SYSTEM DASDA1_27 (* System Configuration *)
  (* Standard: 61499-1 *)
  (* Version 0.4, 2009-03-05, JHC, Holobloc Inc., Deleted Application. *)
  (* Version 0.3, 2003-12-05, JHC, Rockwell Automation, Renamed from NEWSYSTEM. *)
  (* Version 0.2, 2002-11-05, JHC, Rockwell Automation, Fixed missing (empty) FBD in Application. *)
  (* Version 0.1, 2002-01-17, JHC, Rockwell Automation, Minor cleanup *)
  (* Version 0.0, 2000-05-27, JHC, Rockwell Automation *)
  DEVICE HMI_LAYER : FRAME_DEVICE(BOUNDS := [0,0,200,600])
    RESOURCE HMI_left : PANEL_RESOURCE(COLS := 1, ROWS := 10)
      FBS
        start2 : PUBL_0;
        greenTime2 : IN_ANY(TYPE := "UINT", QI := 1, IVAL := "5");
        yellowTime2 : IN_ANY(QI := 1, TYPE := "UINT", IVAL := "1");
        times2 : PUBL_2;
        LABEL1 : FB_LABEL(LABEL := "Western lights control", QI := 1);
        LABEL2 : FB_LABEL(LABEL := "Green time", QI := 1);
        LABEL3 : FB_LABEL(LABEL := "Yellow time", QI := 1);
        minGreenTime2 : IN_ANY(TYPE := "UINT", QI := 1, IVAL := "3");
        LABEL4 : FB_LABEL(LABEL := "Minimum green time", QI := 1);
        Walker1 : IN_EVENT(LABEL := "Walker", QI := 1);
        WalkerTimes2 : PUBL_1;
        RoadControl1 : SUBL_0;
        permit2 : E_PERMIT;
        setreset2 : E_SR;
        split1 : E_SPLIT;
        RoadControl2 : SUBL_0;
        pressCounter : E_CTD(PV := 4);
        split3 : E_SPLIT;
        split4 : E_SPLIT;
        select1 : E_SEL_UINT;
        PedestrianControl2 : SUBL_0;
        gdelay : E_DELAY(DT := t#4000ms);
        setreset3 : E_SR;
        and : FB_AND;
        merge3 : E_MERGE;
        gtrig : E_TRIG;
      END_FBS
      EVENT_CONNECTIONS
        yellowTime2.IND TO times2.REQ;
        LABEL1.INITO TO LABEL2.INIT;
        LABEL2.INITO TO greenTime2.INIT;
        greenTime2.INITO TO LABEL4.INIT;
        LABEL4.INITO TO minGreenTime2.INIT;
        greenTime2.IND TO yellowTime2.REQ;
        yellowTime2.INITO TO times2.INIT;
        times2.INITO TO start2.INIT;
        times2.CNF TO start2.REQ;
        minGreenTime2.INITO TO Walker1.INIT;
        Walker1.INITO TO LABEL3.INIT;
        LABEL3.INITO TO yellowTime2.INIT;
        start2.INITO TO WalkerTimes2.INIT;
        START.COLD TO RoadControl1.INIT;
        RoadControl1.IND TO split1.EI;
        RoadControl2.IND TO setreset2.R;
        RoadControl1.INITO TO RoadControl2.INIT;
        RoadControl2.INITO TO LABEL1.INIT;
        split4.EO1 TO setreset2.S;
        Walker1.IND TO permit2.EI;
        permit2.EO TO split3.EI;
        split3.EO1 TO minGreenTime2.REQ;
        minGreenTime2.IND TO select1.EI0;
        select1.EO TO WalkerTimes2.REQ;
        split4.EO2 TO pressCounter.LD;
        split3.EO2 TO pressCounter.CD;
        PedestrianControl2.IND TO gdelay.START;
        gdelay.EO TO setreset3.S;
        setreset3.EO TO merge3.EI1;
        pressCounter.CDO TO merge3.EI2;
        merge3.EO TO and.REQ;
        and.CNF TO gtrig.EI;
        gtrig.ER TO select1.EI1;
        gtrig.EF TO setreset3.R;
        split1.EO1 TO greenTime2.REQ;
        split1.EO2 TO split4.EI;
        WalkerTimes2.INITO TO PedestrianControl2.INIT;
      END_CONNECTIONS
      DATA_CONNECTIONS
        yellowTime2.OUT TO times2.SD_2;
        greenTime2.OUT TO times2.SD_1;
        setreset2.Q TO permit2.PERMIT;
        minGreenTime2.OUT TO select1.IN0;
        select1.OUT TO WalkerTimes2.SD_1;
        pressCounter.CV TO select1.IN1;
        setreset3.Q TO and.IN1;
        pressCounter.Q TO and.IN2;
        and.OUT TO gtrig.QI;
      END_CONNECTIONS
    END_RESOURCE
    RESOURCE HMI_up : PANEL_RESOURCE(COLS := 1, ROWS := 10)
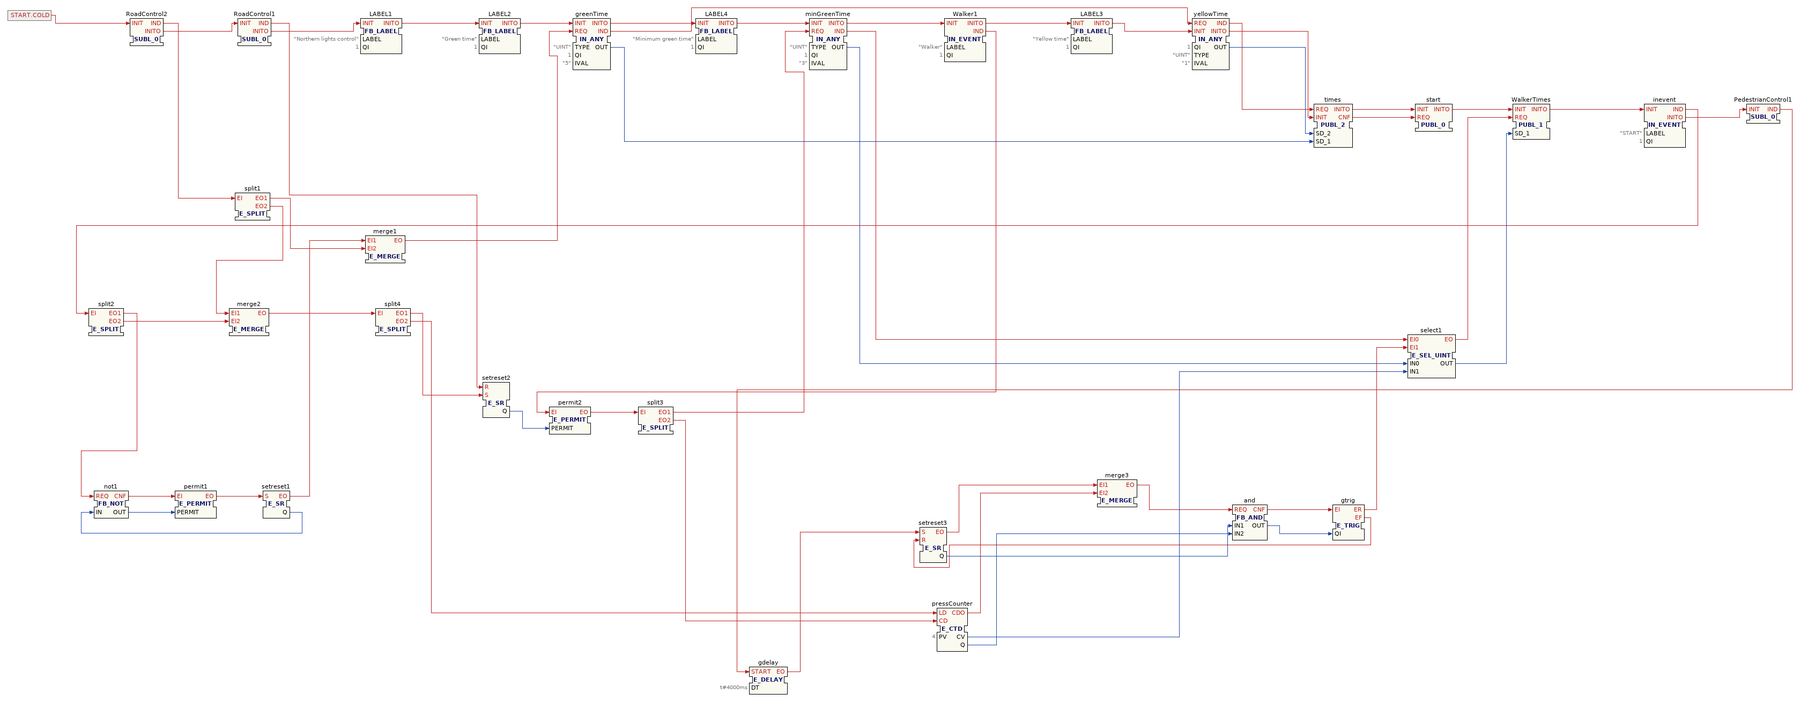
      FBS
        start : PUBL_0;
        greenTime : IN_ANY(TYPE := "UINT", QI := 1, IVAL := "5");
        yellowTime : IN_ANY(QI := 1, TYPE := "UINT", IVAL := "1");
        times : PUBL_2;
        LABEL1 : FB_LABEL(LABEL := "Northern lights control", QI := 1);
        LABEL2 : FB_LABEL(LABEL := "Green time", QI := 1);
        LABEL3 : FB_LABEL(LABEL := "Yellow time", QI := 1);
        minGreenTime : IN_ANY(TYPE := "UINT", QI := 1, IVAL := "3");
        LABEL4 : FB_LABEL(LABEL := "Minimum green time", QI := 1);
        Walker1 : IN_EVENT(LABEL := "Walker", QI := 1);
        WalkerTimes : PUBL_1;
        inevent : IN_EVENT(LABEL := "START", QI := 1);
        RoadControl2 : SUBL_0;
        merge1 : E_MERGE;
        permit1 : E_PERMIT;
        setreset1 : E_SR;
        not1 : FB_NOT;
        permit2 : E_PERMIT;
        setreset2 : E_SR;
        split1 : E_SPLIT;
        RoadControl1 : SUBL_0;
        merge2 : E_MERGE;
        split2 : E_SPLIT;
        pressCounter : E_CTD(PV := 4);
        split3 : E_SPLIT;
        split4 : E_SPLIT;
        select1 : E_SEL_UINT;
        PedestrianControl1 : SUBL_0;
        gdelay : E_DELAY(DT := t#4000ms);
        setreset3 : E_SR;
        and : FB_AND;
        merge3 : E_MERGE;
        gtrig : E_TRIG;
      END_FBS
      EVENT_CONNECTIONS
        yellowTime.IND TO times.REQ;
        LABEL1.INITO TO LABEL2.INIT;
        LABEL2.INITO TO greenTime.INIT;
        greenTime.INITO TO LABEL4.INIT;
        LABEL4.INITO TO minGreenTime.INIT;
        greenTime.IND TO yellowTime.REQ;
        yellowTime.INITO TO times.INIT;
        times.INITO TO start.INIT;
        times.CNF TO start.REQ;
        minGreenTime.INITO TO Walker1.INIT;
        Walker1.INITO TO LABEL3.INIT;
        LABEL3.INITO TO yellowTime.INIT;
        start.INITO TO WalkerTimes.INIT;
        merge1.EO TO greenTime.REQ;
        not1.CNF TO permit1.EI;
        permit1.EO TO setreset1.S;
        setreset1.EO TO merge1.EI1;
        START.COLD TO RoadControl2.INIT;
        WalkerTimes.INITO TO inevent.INIT;
        RoadControl2.IND TO split1.EI;
        split1.EO1 TO merge1.EI2;
        RoadControl1.IND TO setreset2.R;
        RoadControl2.INITO TO RoadControl1.INIT;
        RoadControl1.INITO TO LABEL1.INIT;
        split1.EO2 TO merge2.EI1;
        inevent.IND TO split2.EI;
        split2.EO1 TO not1.REQ;
        split2.EO2 TO merge2.EI2;
        merge2.EO TO split4.EI;
        split4.EO1 TO setreset2.S;
        Walker1.IND TO permit2.EI;
        permit2.EO TO split3.EI;
        split3.EO1 TO minGreenTime.REQ;
        minGreenTime.IND TO select1.EI0;
        select1.EO TO WalkerTimes.REQ;
        split4.EO2 TO pressCounter.LD;
        split3.EO2 TO pressCounter.CD;
        inevent.INITO TO PedestrianControl1.INIT;
        PedestrianControl1.IND TO gdelay.START;
        gdelay.EO TO setreset3.S;
        setreset3.EO TO merge3.EI1;
        pressCounter.CDO TO merge3.EI2;
        merge3.EO TO and.REQ;
        and.CNF TO gtrig.EI;
        gtrig.ER TO select1.EI1;
        gtrig.EF TO setreset3.R;
      END_CONNECTIONS
      DATA_CONNECTIONS
        yellowTime.OUT TO times.SD_2;
        greenTime.OUT TO times.SD_1;
        not1.OUT TO permit1.PERMIT;
        setreset1.Q TO not1.IN;
        setreset2.Q TO permit2.PERMIT;
        minGreenTime.OUT TO select1.IN0;
        select1.OUT TO WalkerTimes.SD_1;
        pressCounter.CV TO select1.IN1;
        setreset3.Q TO and.IN1;
        pressCounter.Q TO and.IN2;
        and.OUT TO gtrig.QI;
      END_CONNECTIONS
    END_RESOURCE
  END_DEVICE
  DEVICE MODEL_LAYER : FRAME_DEVICE
    RESOURCE LIGHTS_U : PANEL_RESOURCE
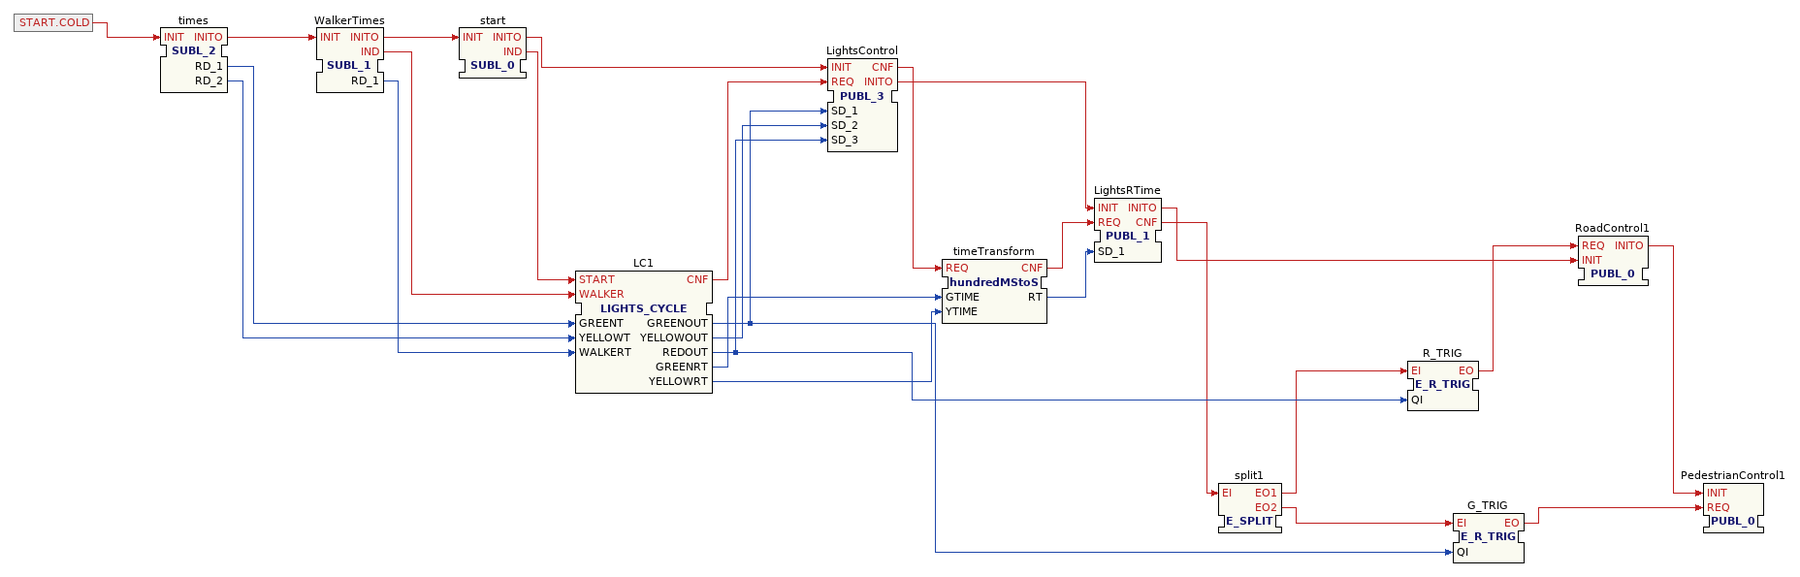
      FBS
        LightsControl : PUBL_3;
        start : SUBL_0;
        times : SUBL_2;
        WalkerTimes : SUBL_1;
        LC1 : LIGHTS_CYCLE;
        R_TRIG : E_R_TRIG;
        RoadControl1 : PUBL_0;
        timeTransform : hundredMStoS;
        LightsRTime : PUBL_1;
        G_TRIG : E_R_TRIG;
        PedestrianControl1 : PUBL_0;
        split1 : E_SPLIT;
      END_FBS
      EVENT_CONNECTIONS
        START.COLD TO times.INIT;
        start.INITO TO LightsControl.INIT;
        times.INITO TO WalkerTimes.INIT;
        WalkerTimes.INITO TO start.INIT;
        start.IND TO LC1.START;
        WalkerTimes.IND TO LC1.WALKER;
        LC1.CNF TO LightsControl.REQ;
        R_TRIG.EO TO RoadControl1.REQ;
        LightsControl.CNF TO timeTransform.REQ;
        LightsControl.INITO TO LightsRTime.INIT;
        LightsRTime.INITO TO RoadControl1.INIT;
        timeTransform.CNF TO LightsRTime.REQ;
        RoadControl1.INITO TO PedestrianControl1.INIT;
        G_TRIG.EO TO PedestrianControl1.REQ;
        LightsRTime.CNF TO split1.EI;
        split1.EO1 TO R_TRIG.EI;
        split1.EO2 TO G_TRIG.EI;
      END_CONNECTIONS
      DATA_CONNECTIONS
        WalkerTimes.RD_1 TO LC1.WALKERT;
        times.RD_1 TO LC1.GREENT;
        times.RD_2 TO LC1.YELLOWT;
        LC1.GREENOUT TO LightsControl.SD_1;
        LC1.YELLOWOUT TO LightsControl.SD_2;
        LC1.REDOUT TO LightsControl.SD_3;
        LC1.REDOUT TO R_TRIG.QI;
        LC1.GREENRT TO timeTransform.GTIME;
        LC1.YELLOWRT TO timeTransform.YTIME;
        timeTransform.RT TO LightsRTime.SD_1;
        LC1.GREENOUT TO G_TRIG.QI;
      END_CONNECTIONS
    END_RESOURCE
    RESOURCE LIGHTS_L : PANEL_RESOURCE
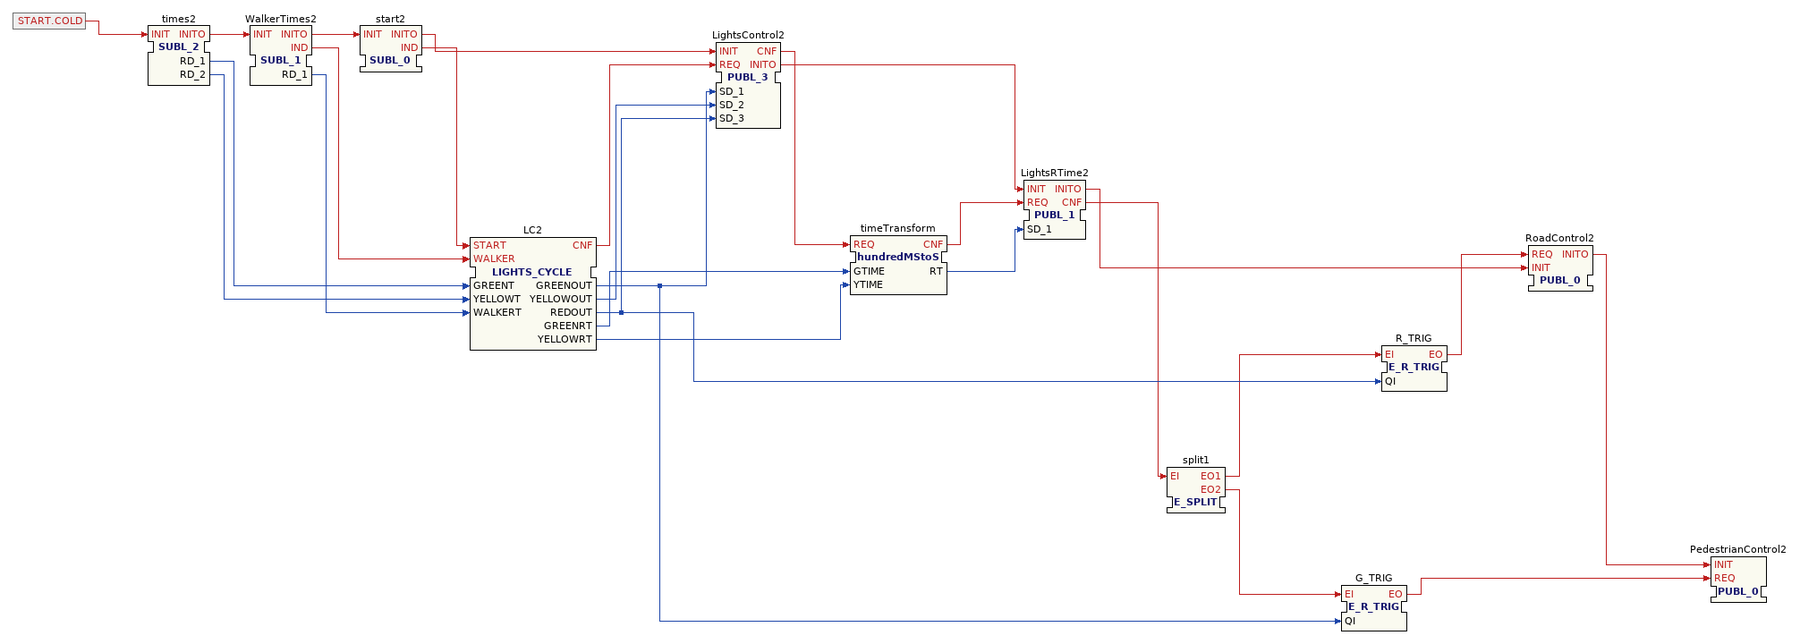
      FBS
        LightsControl2 : PUBL_3;
        start2 : SUBL_0;
        times2 : SUBL_2;
        WalkerTimes2 : SUBL_1;
        LC2 : LIGHTS_CYCLE;
        R_TRIG : E_R_TRIG;
        RoadControl2 : PUBL_0;
        timeTransform : hundredMStoS;
        LightsRTime2 : PUBL_1;
        PedestrianControl2 : PUBL_0;
        split1 : E_SPLIT;
        G_TRIG : E_R_TRIG;
      END_FBS
      EVENT_CONNECTIONS
        START.COLD TO times2.INIT;
        start2.INITO TO LightsControl2.INIT;
        times2.INITO TO WalkerTimes2.INIT;
        WalkerTimes2.INITO TO start2.INIT;
        start2.IND TO LC2.START;
        WalkerTimes2.IND TO LC2.WALKER;
        LC2.CNF TO LightsControl2.REQ;
        R_TRIG.EO TO RoadControl2.REQ;
        LightsControl2.CNF TO timeTransform.REQ;
        LightsControl2.INITO TO LightsRTime2.INIT;
        LightsRTime2.INITO TO RoadControl2.INIT;
        timeTransform.CNF TO LightsRTime2.REQ;
        LightsRTime2.CNF TO split1.EI;
        split1.EO1 TO R_TRIG.EI;
        split1.EO2 TO G_TRIG.EI;
        RoadControl2.INITO TO PedestrianControl2.INIT;
        G_TRIG.EO TO PedestrianControl2.REQ;
      END_CONNECTIONS
      DATA_CONNECTIONS
        WalkerTimes2.RD_1 TO LC2.WALKERT;
        times2.RD_1 TO LC2.GREENT;
        times2.RD_2 TO LC2.YELLOWT;
        LC2.GREENOUT TO LightsControl2.SD_1;
        LC2.YELLOWOUT TO LightsControl2.SD_2;
        LC2.REDOUT TO LightsControl2.SD_3;
        LC2.REDOUT TO R_TRIG.QI;
        LC2.GREENRT TO timeTransform.GTIME;
        LC2.YELLOWRT TO timeTransform.YTIME;
        timeTransform.RT TO LightsRTime2.SD_1;
        LC2.GREENOUT TO G_TRIG.QI;
      END_CONNECTIONS
    END_RESOURCE
  END_DEVICE
  DEVICE VIEW_LAYER : FRAME_DEVICE(BOUNDS := [200,0,630,400], GRID := [1,1])
    RESOURCE view_res : PANEL_RESOURCE
      FBS
        LightsControl : SUBL_3;
        GREENVIEW : OUT_BOOL(C0 := [255,255,255], C1 := [0,255,0], QI := 1, LABEL := " ");
        YELLOWVIEW : OUT_BOOL(C0 := [255,255,255], C1 := [255,255,0], QI := 1, LABEL := " ");
        REDVIEW : OUT_BOOL(C0 := [255,255,255], C1 := [255,0,0], QI := 1, LABEL := " ");
        space11 : XSPACE(DIA := 1, DIMS := [220,75]);
        space12 : XSPACE(DIA := 1, DIMS := [10,75], COLORS := [black,black]);
        space13 : XSPACE(DIA := 1, DIMS := [40,75]);
        space16 : XSPACE(DIA := 1, DIMS := [10,75], COLORS := [black,black]);
        space17 : XSPACE(DIA := 1, DIMS := [220,75]);
        space21 : XSPACE(DIA := 1, DIMS := [220,25]);
        space22 : XSPACE(DIA := 1, DIMS := [10,25], COLORS := [black,black]);
        space23 : XSPACE(DIA := 1, DIMS := [40,25]);
        space24 : XSPACE(DIMS := [38,25], DIA := 1);
        space25 : XSPACE(DIMS := [10,25], DIA := 1, COLORS := [black,black]);
        space14 : XSPACE(DIA := 1, DIMS := [30,75], LBLS := "RT:, , , , ");
        RT : OUT_ANY(QI := 1, TYPE := "UINT", W := 3);
        space15 : XSPACE(DIA := 1, DIMS := [40,75]);
        space26 : XSPACE(DIMS := [200,25], DIA := 1);
        space31 : XSPACE(DIMS := [230,10], DIA := 1, COLORS := [black,black]);
        space32 : XSPACE(DIMS := [147,10], DIA := 1);
        space33 : XSPACE(DIMS := [220,10], DIA := 1, COLORS := [black,black]);
        space41 : XSPACE(DIMS := [595,40], DIA := 1);
        space42 : XSPACE(DIMS := [180,20], DIA := 1);
        LightsControl2 : SUBL_3;
        GREENVIEW2 : OUT_BOOL(C0 := [255,255,255], C1 := [0,255,0], QI := 1, LABEL := " ");
        space43 : XSPACE(DIMS := [400,20], DIA := 1);
        space51 : XSPACE(DIMS := [100,20], DIA := 1, LBLS := " , ,RT: , , ");
        RT2 : OUT_ANY(QI := 1, TYPE := "UINT", W := 3);
        space52 : XSPACE(DIMS := [43,20], DIA := 1);
        YELLOWVIEW2 : OUT_BOOL(C0 := [255,255,255], C1 := [255,255,0], QI := 1, LABEL := " ");
        space53 : XSPACE(DIMS := [400,20], DIA := 1);
        space61 : XSPACE(DIMS := [180,20], DIA := 1);
        REDVIEW2 : OUT_BOOL(C0 := [255,255,255], C1 := [255,0,0], QI := 1, LABEL := " ");
        space62 : XSPACE(DIMS := [400,20], DIA := 1);
        space71 : XSPACE(DIMS := [595,40], DIA := 1);
        space81 : XSPACE(DIMS := [230,10], DIA := 1, COLORS := [black,black]);
        space82 : XSPACE(DIMS := [147,10], DIA := 1);
        space83 : XSPACE(DIMS := [220,10], DIA := 1, COLORS := [black,black]);
        space91 : XSPACE(DIMS := [220,75], DIA := 1);
        space92 : XSPACE(DIMS := [10,75], DIA := 1, COLORS := [black,black]);
        space93 : XSPACE(DIMS := [147,75], DIA := 1);
        space94 : XSPACE(DIMS := [10,75], DIA := 1, COLORS := [black,black]);
        LightsRTime : SUBL_1;
        LightsRTime2 : SUBL_1;
      END_FBS
      EVENT_CONNECTIONS
        LightsControl.INITO TO GREENVIEW.INIT;
        GREENVIEW.INITO TO YELLOWVIEW.INIT;
        YELLOWVIEW.INITO TO REDVIEW.INIT;
        LightsControl.IND TO GREENVIEW.REQ;
        GREENVIEW.CNF TO YELLOWVIEW.REQ;
        YELLOWVIEW.CNF TO REDVIEW.REQ;
        START.COLD TO space11.INIT;
        space11.INITO TO space12.INIT;
        space12.INITO TO space13.INIT;
        space16.INITO TO space17.INIT;
        space17.INITO TO space21.INIT;
        space21.INITO TO space22.INIT;
        space22.INITO TO space23.INIT;
        space23.INITO TO LightsControl.INIT;
        REDVIEW.INITO TO space24.INIT;
        space24.INITO TO space25.INIT;
        space13.INITO TO space14.INIT;
        RT.INITO TO space15.INIT;
        space15.INITO TO space16.INIT;
        space25.INITO TO space26.INIT;
        space26.INITO TO space31.INIT;
        space31.INITO TO space32.INIT;
        space32.INITO TO space33.INIT;
        space33.INITO TO space41.INIT;
        space41.INITO TO space42.INIT;
        space42.INITO TO LightsControl2.INIT;
        LightsControl2.INITO TO GREENVIEW2.INIT;
        LightsControl2.IND TO GREENVIEW2.REQ;
        GREENVIEW2.INITO TO space43.INIT;
        space43.INITO TO space51.INIT;
        RT2.INITO TO space52.INIT;
        space52.INITO TO YELLOWVIEW2.INIT;
        YELLOWVIEW2.INITO TO space53.INIT;
        space53.INITO TO space61.INIT;
        space61.INITO TO REDVIEW2.INIT;
        REDVIEW2.INITO TO space62.INIT;
        space62.INITO TO space71.INIT;
        space71.INITO TO space81.INIT;
        space81.INITO TO space82.INIT;
        space82.INITO TO space83.INIT;
        space83.INITO TO space91.INIT;
        space91.INITO TO space92.INIT;
        space92.INITO TO space93.INIT;
        space93.INITO TO space94.INIT;
        GREENVIEW2.CNF TO YELLOWVIEW2.REQ;
        YELLOWVIEW2.CNF TO REDVIEW2.REQ;
        space14.INITO TO LightsRTime.INIT;
        LightsRTime.INITO TO RT.INIT;
        LightsRTime.IND TO RT.REQ;
        space51.INITO TO LightsRTime2.INIT;
        LightsRTime2.INITO TO RT2.INIT;
        LightsRTime2.IND TO RT2.REQ;
      END_CONNECTIONS
      DATA_CONNECTIONS
        LightsControl.RD_1 TO GREENVIEW.IN;
        LightsControl.RD_2 TO YELLOWVIEW.IN;
        LightsControl.RD_3 TO REDVIEW.IN;
        LightsControl2.RD_1 TO GREENVIEW2.IN;
        LightsControl2.RD_2 TO YELLOWVIEW2.IN;
        LightsControl2.RD_3 TO REDVIEW2.IN;
        LightsRTime.RD_1 TO RT.IN;
        LightsRTime2.RD_1 TO RT2.IN;
      END_CONNECTIONS
    END_RESOURCE
  END_DEVICE
END_SYSTEM
